# EPICS substitutions: bkhApp/Db/bkh11.substitutions
file analogIn.db
{
pattern { N,ADDR,  DESC,      MOD,  PORT, EGU,EOFF,       ESLO,PREC}
	{ 1,   0,Chan01,3408-$(M), A3408,   V,   0,0.000305185,   2}
	{ 2,   1,Chan02,3408-$(M), A3408,   V,   0,0.000305185,   2}
	{ 3,   2,Chan03,3408-$(M), A3408,   V,   0,0.000305185,   2}
	{ 4,   3,Chan04,3408-$(M), A3408,   V,   0,0.000305185,   2}
	{ 5,   4,Chan05,3408-$(M), A3408,   V,   0,0.000305185,   2}
	{ 6,   5,Chan06,3408-$(M), A3408,   V,   0,0.000305185,   2}
	{ 7,   6,Chan07,3408-$(M), A3408,   V,   0,0.000305185,   2}
	{ 8,   7,Chan08,3408-$(M), A3408,   V,   0,0.000305185,   2}
}
file analogTemp.db
{
pattern { N,ADDR,  DESC, MOD,  PORT, ESLO,PREC}
	{ 1,   0,Chan01,3314, A3314,  0.1,   2}
	{ 2,   1,Chan02,3314, A3314,  0.1,   2}
	{ 3,   2,Chan03,3314, A3314,  0.1,   2}
	{ 4,   3,Chan04,3314, A3314,  0.1,   2}
}
file bkhBo.db
{
pattern	{ N,       MOD,  PORT, OFF}
	{ 1, 2114-$(M), A2114,   0}
	{ 2, 2114-$(M), A2114,   1}
	{ 3, 2114-$(M), A2114,   2}
	{ 4, 2114-$(M), A2114,   3}
	{ 5, 2114-$(M), A2114,   4}
	{ 6, 2114-$(M), A2114,   5}
	{ 7, 2114-$(M), A2114,   6}
	{ 8, 2114-$(M), A2114,   7}

	{ 1, 2124-$(M), A2124,   0}
	{ 2, 2124-$(M), A2124,   1}
	{ 3, 2124-$(M), A2124,   2}
	{ 4, 2124-$(M), A2124,   3}
	{ 5, 2124-$(M), A2124,   4}
	{ 6, 2124-$(M), A2124,   5}
	{ 7, 2124-$(M), A2124,   6}
	{ 8, 2124-$(M), A2124,   7}
}
file readwrite.db
{
pattern	{      MOD,  PORT}
	{3408-$(M), A3408}
	{3314-$(M), A3314}
}
file bkhAdrv.db
{
pattern	{      MOD,  PORT}
	{3408-$(M), A3408}
	{3314-$(M), A3314}
	{2114-$(M), A2114}
	{2124-$(M), A2124}
}
file bkhAErr.db
{
pattern	{      MOD,  PORT}
	{3408-$(M), A3408}
	{3314-$(M), A3314}
}
file b9000.db{
	{ RPORT=B900R, WPORT=B900W}
}
file b9000RRegs.db
{
pattern	{ N,                 DESC,  PORT}
	{10,      "PLC Interface", B900R}
	{11, "Bus Term Diagnossi", B900R}
	{12, "Bus Coupler Status", B900R}
	{16, "anlg output length", B900R}
	{17, "anlg inputs length", B900R}
	{18, "Outpt Image length", B900R}
	{19, "Input Image length", B900R}
	{32, "Watchdog curr time", B900R}
}
file b9000WRegs.db
{
pattern	{ N,                 DESC,  PORT}
	{ 0,      "PLC Interface", B900W}
	{ 1, "Bus Term Diagnossi", B900W}
	{22,"Watchdog Tmout (ms)", B900W}
	{23,     "Watchdog Reset", B900W}
	{24,      "Watchdog type", B900W}
	{25,    "Modbus TCP mode", B900W}
}
